Staubli VAL3: OUT.dtx

public string sItems
string sMessage
string sKey
